{attribute 'linkalways'} 
{attribute 'no_explicit_call' := 'This FB is a CLASS and must be accessed using methods or properties'}
{attribute 'enable_dynamic_creation'}
FUNCTION_BLOCK FINAL ABS_UDINT EXTENDS Node
VAR
	in : _UDINT(0);
	out : _UDINT(0);
END_VAR

METHOD PUBLIC Clone : I_Node
VAR
	pNode : POINTER TO ABS_UDINT;
END_VAR
pNode := __NEW(ABS_UDINT);
Clone := pNode^;
END_METHOD

METHOD FB_init : BOOL
VAR_INPUT
	bInitRetains : BOOL; // if TRUE, the retain variables are initialized (warm start / cold start)
	bInCopyCode : BOOL;  // if TRUE, the instance afterwards gets moved into the copy code (online change)
END_VAR
AddInput('in',THIS^.in);
AddOutput('out', THIS^.out);
END_METHOD

METHOD PROTECTED OnExecute
VAR
END_VAR
out.Value := ABS(in.Value);
END_METHOD

END_FUNCTION_BLOCK

(* stored: Version 1.1.0.1, ProductVersion 3.1.4024.15
   POU ABS_UDINT: Id {a2d7947f-eb56-4aac-96f1-24b3a568bdc6}, SpecialFunc None
   Folder Constructor: Id {f64083ee-5750-43c1-8c5d-d8034d99f4d2}
   Method Clone: Id {0a7db46b-6033-4a5f-919b-51fcb61d9731}
   Method FB_init: Id {a6880978-0d6a-43fe-a81b-f7c55a62872f}
   Method OnExecute: Id {e9f26671-363c-4da3-a530-5926d7f8b158} *)
